// TIA Portal V17 export
// export: Created 2024-08-07T21:44:12.1713067Z, ExportSetting WithDefaults, DisplayName Totally Integrated Automation Portal, DisplayVersion V17 Update 7, DisplayName TIA Portal Openness, DisplayVersion V17 Update 7, DisplayName TIA Portal Version Control Interface, DisplayVersion V17, DisplayName SINAMICS Startdrive Advanced, DisplayVersion V17 SP2, DisplayName SINAMICS Startdrive G110M, G120, G120C, G120D, G120P, G115D, DisplayVersion V17 SP2, DisplayName SINAMICS Startdrive G130, G150, S120, S150, SINAMICS MV, S210, DisplayVersion V17 SP2, DisplayName STEP 7 Professional, DisplayVersion V17 Update 7, DisplayName STEP 7 Safety, DisplayVersion V17 Update 6, DisplayName WinCC Advanced / Unified PC, DisplayVersion V17 Update 7
VAR_GLOBAL   // PLC tag table "Default tag table"
   tAirPressureOK AT %T0 : Timer;
   "ALARMA ACTIVA" AT %M6.0 : Bool;
   ALARMA_2 AT %MW8 : Int;
   ALARMA_3 AT %MW10 : Int;
   ALARMA_4 AT %MW12 : Int;
   ALARMA_5 AT %MW14 : Int;
   ALARM_AKCNOWLEDGE AT %M6.1 : Bool;
   INIT_SCAN AT %M6.2 : Bool;
END_VAR
VAR_GLOBAL CONSTANT   // user constants
   NumberOfEksKeys : Int := 100;
   NumberOfEksEngineerKeys : Int := 5;
   GapLeaderLevel : Int := 2;
   MaintenanceLevel : Int := 3;
   EngineerLevel : Int := 5;
   NumberOfProductionPrograms : UInt := 8;
   NumberOfProductionProducts : Int := 8;
   LoggerBufferSize : Int := 32;
   LoggerTypeAlarm : Int := 1;
   LoggerTypeStatus : Int := 2;
   LoggerNumberOfPartErrors : Int := 5;
   LoggerTypePart : Int := 3;
   LoggerTypeUser : Int := 4;
   LoggerTypeComment : Int := 99;
   AlarmsCount : Int := 256;
   NumberOfIJCoreMessages : Int := 30;
   LoggerTypeRiveting : Int := 50;
   EksNumberOfKeys : Int := 100;
   EksNumberOfEngineerKeys : Int := 50;
   EksGapLeaderLevel : Int := 2;
   EksMaintenanceLevel : Int := 3;
   EksEngineerLevel : Int := 5;
END_VAR
